// TIA Portal V16 export
// export: Created 2023-03-29T11:03:22.8937911Z, ExportSetting WithDefaults, DisplayName Totally Integrated Automation Portal, DisplayVersion V16 Update 6, DisplayName TIA Portal Version Control Interface, DisplayVersion V16 Update 2, DisplayName TIA Portal Openness, DisplayVersion V16 Update 6, DisplayName STEP 7 Professional, DisplayVersion V16 Update 6, DisplayName STEP 7 Safety, DisplayVersion V16, DisplayName WinCC Advanced, DisplayVersion V16 Update 6
FUNCTION "Wybór_aktywnego_zbiornika" : Void   // FC20, LAD
TITLE = Compressor selection from hours
{ S7_Optimized_Access := 'TRUE' }
AUTHOR : rtecmer
VERSION : 0.1
// Ustawienie kolejności wyboru zbiornika z wyrównaniem czasu pracy. Podstawa najmniejsza ilość godzin pracy
// stored: AutoNumber true, IsIECCheckEnabled false, SetENOAutomatically false, UDAEnableTagReadback false
   VAR_INPUT
      aktywny_Zbiornik_1 : Bool;   // zbiornik aktywny zasuwy na pozycji atomat
      aktywny_Zbiornik_2 : Bool;
      aktywny_Zbiornik_3 : Bool;
      aktywny_Zbiornik_4 : Bool;
      ready_Z1 : Bool;   // gotowość
      ready_Z2 : Bool;   // gotowość
      ready_Z3 : Bool;   // gotowość
      ready_Z4 : Bool;   // gotowość
      ready_Z5 : Bool;   // gotowość
      ready_Z6 : Bool;   // gotowość
      ready_Z7 : Bool;   // gotowość
      ready_Z8 : Bool;   // gotowość
      Is_Eptying : Bool;   // aktwny cykl napełniania
      Is_Filling : Bool;   // aktywny cykl pompownia
   END_VAR
   VAR_IN_OUT
      Reset : Bool;   // Reset po błędzie
      set_HWork_Tank_1 : Bool;   // ustawiony aktywny
      set_HWork_Tank_2 : Bool;   // ustawiony aktywny
      set_HWork_Tank_3 : Bool;   // ustawiony aktywny
      set_HWork_Tank_4 : Bool;   // ustawiony aktywny
      blok_tank_1 : Bool;   // blokowanie zbirnika w sekwencji
      blok_tank_2 : Bool;   // blokowanie zbirnika w sekwencji
      blok_tank_3 : Bool;   // blokowanie zbirnika w sekwencji
      blok_tank_4 : Bool;   // blokowanie zbirnika w sekwencji
   END_VAR
   VAR_TEMP
      tmp_Sum_sek_P1 : Real;
      tmp_Sum_sek_P2 : Real;
      tmp_Sum_sek_P3 : Real;
      tmp_Sum_sek_P4 : Real;
   END_VAR
BEGIN

REGION Network 1: Reakcja na równe liczniki
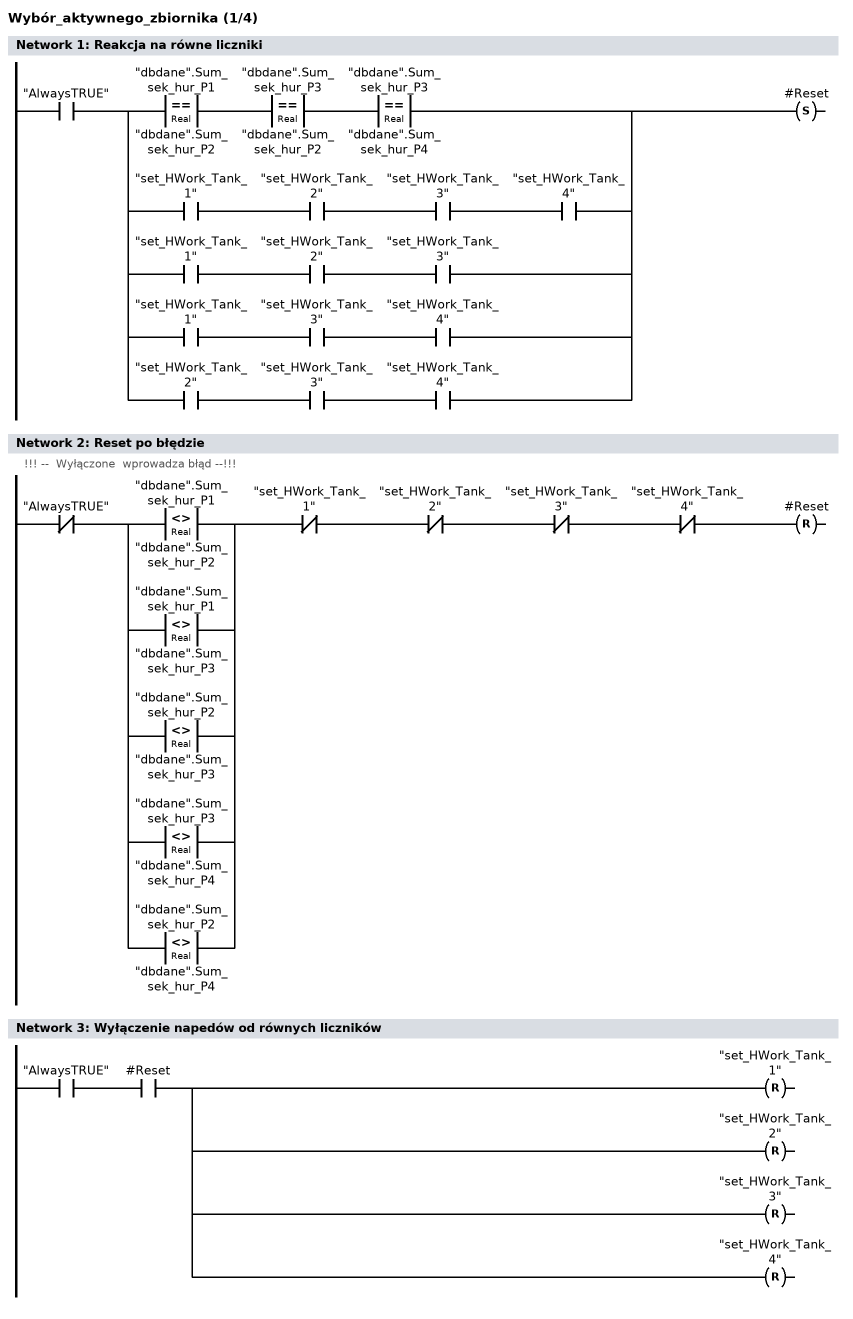
   RUNG wire#powerrail
      Contact( "AlwaysTRUE" )
      wire#w1
      { S7_Templates := "SrcType := Real" } EQ_Contact(in1 := "dbdane".Sum_sek_hur_P1, in2 := "dbdane".Sum_sek_hur_P2)
      { S7_Templates := "SrcType := Real" } EQ_Contact(in1 := "dbdane".Sum_sek_hur_P3, in2 := "dbdane".Sum_sek_hur_P2)
      { S7_Templates := "SrcType := Real" } EQ_Contact(in1 := "dbdane".Sum_sek_hur_P3, in2 := "dbdane".Sum_sek_hur_P4)
      wire#w2
      S_Coil( #Reset )
   END_RUNG
   RUNG wire#w1
      Contact( "set_HWork_Tank_1" )
      Contact( "set_HWork_Tank_2" )
      Contact( "set_HWork_Tank_3" )
      Contact( "set_HWork_Tank_4" )
   END_RUNG wire#w2
   RUNG wire#w1
      Contact( "set_HWork_Tank_1" )
      Contact( "set_HWork_Tank_2" )
      Contact( "set_HWork_Tank_3" )
   END_RUNG wire#w2
   RUNG wire#w1
      Contact( "set_HWork_Tank_1" )
      Contact( "set_HWork_Tank_3" )
      Contact( "set_HWork_Tank_4" )
   END_RUNG wire#w2
   RUNG wire#w1
      Contact( "set_HWork_Tank_2" )
      Contact( "set_HWork_Tank_3" )
      Contact( "set_HWork_Tank_4" )
   END_RUNG wire#w2
   // the same network as SCL:
   IF "AlwaysTRUE" AND ((("dbdane".Sum_sek_hur_P1 = "dbdane".Sum_sek_hur_P2) AND ("dbdane".Sum_sek_hur_P3 = "dbdane".Sum_sek_hur_P2) AND ("dbdane".Sum_sek_hur_P3 = "dbdane".Sum_sek_hur_P4)) OR ("set_HWork_Tank_1" AND "set_HWork_Tank_2" AND "set_HWork_Tank_3" AND "set_HWork_Tank_4") OR ("set_HWork_Tank_1" AND "set_HWork_Tank_2" AND "set_HWork_Tank_3") OR ("set_HWork_Tank_1" AND "set_HWork_Tank_3" AND "set_HWork_Tank_4") OR ("set_HWork_Tank_2" AND "set_HWork_Tank_3" AND "set_HWork_Tank_4")) THEN
       #Reset := TRUE;
   END_IF;
END_REGION

REGION Network 2: Reset po błędzie
   // !!! --  Wyłączone  wprowadza błąd --!!!
   RUNG wire#powerrail
      I_Contact( "AlwaysTRUE" )
      wire#w1
      { S7_Templates := "SrcType := Real" } NE_Contact(in1 := "dbdane".Sum_sek_hur_P1, in2 := "dbdane".Sum_sek_hur_P2)
      wire#w2
      I_Contact( "set_HWork_Tank_1" )
      I_Contact( "set_HWork_Tank_2" )
      I_Contact( "set_HWork_Tank_3" )
      I_Contact( "set_HWork_Tank_4" )
      R_Coil( #Reset )
   END_RUNG
   RUNG wire#w1
      { S7_Templates := "SrcType := Real" } NE_Contact(in1 := "dbdane".Sum_sek_hur_P1, in2 := "dbdane".Sum_sek_hur_P3)
   END_RUNG wire#w2
   RUNG wire#w1
      { S7_Templates := "SrcType := Real" } NE_Contact(in1 := "dbdane".Sum_sek_hur_P2, in2 := "dbdane".Sum_sek_hur_P3)
   END_RUNG wire#w2
   RUNG wire#w1
      { S7_Templates := "SrcType := Real" } NE_Contact(in1 := "dbdane".Sum_sek_hur_P3, in2 := "dbdane".Sum_sek_hur_P4)
   END_RUNG wire#w2
   RUNG wire#w1
      { S7_Templates := "SrcType := Real" } NE_Contact(in1 := "dbdane".Sum_sek_hur_P2, in2 := "dbdane".Sum_sek_hur_P4)
   END_RUNG wire#w2
   // the same network as SCL:
   IF NOT "AlwaysTRUE" AND (("dbdane".Sum_sek_hur_P1 <> "dbdane".Sum_sek_hur_P2) OR ("dbdane".Sum_sek_hur_P1 <> "dbdane".Sum_sek_hur_P3) OR ("dbdane".Sum_sek_hur_P2 <> "dbdane".Sum_sek_hur_P3) OR ("dbdane".Sum_sek_hur_P3 <> "dbdane".Sum_sek_hur_P4) OR ("dbdane".Sum_sek_hur_P2 <> "dbdane".Sum_sek_hur_P4)) AND NOT "set_HWork_Tank_1" AND NOT "set_HWork_Tank_2" AND NOT "set_HWork_Tank_3" AND NOT "set_HWork_Tank_4" THEN
       #Reset := FALSE;
   END_IF;
END_REGION

REGION Network 3: Wyłączenie napedów od równych liczników
   RUNG wire#powerrail
      Contact( "AlwaysTRUE" )
      Contact( #Reset )
      wire#w1
      R_Coil( "set_HWork_Tank_1" )
   END_RUNG
   RUNG wire#w1
      R_Coil( "set_HWork_Tank_2" )
   END_RUNG
   RUNG wire#w1
      R_Coil( "set_HWork_Tank_3" )
   END_RUNG
   RUNG wire#w1
      R_Coil( "set_HWork_Tank_4" )
   END_RUNG
   // the same network as SCL:
   IF "AlwaysTRUE" AND #Reset THEN
       "set_HWork_Tank_1" := FALSE;
       "set_HWork_Tank_2" := FALSE;
       "set_HWork_Tank_3" := FALSE;
       "set_HWork_Tank_4" := FALSE;
   END_IF;
END_REGION

REGION Network 4: Ustawienie domyślnych liczników startowych
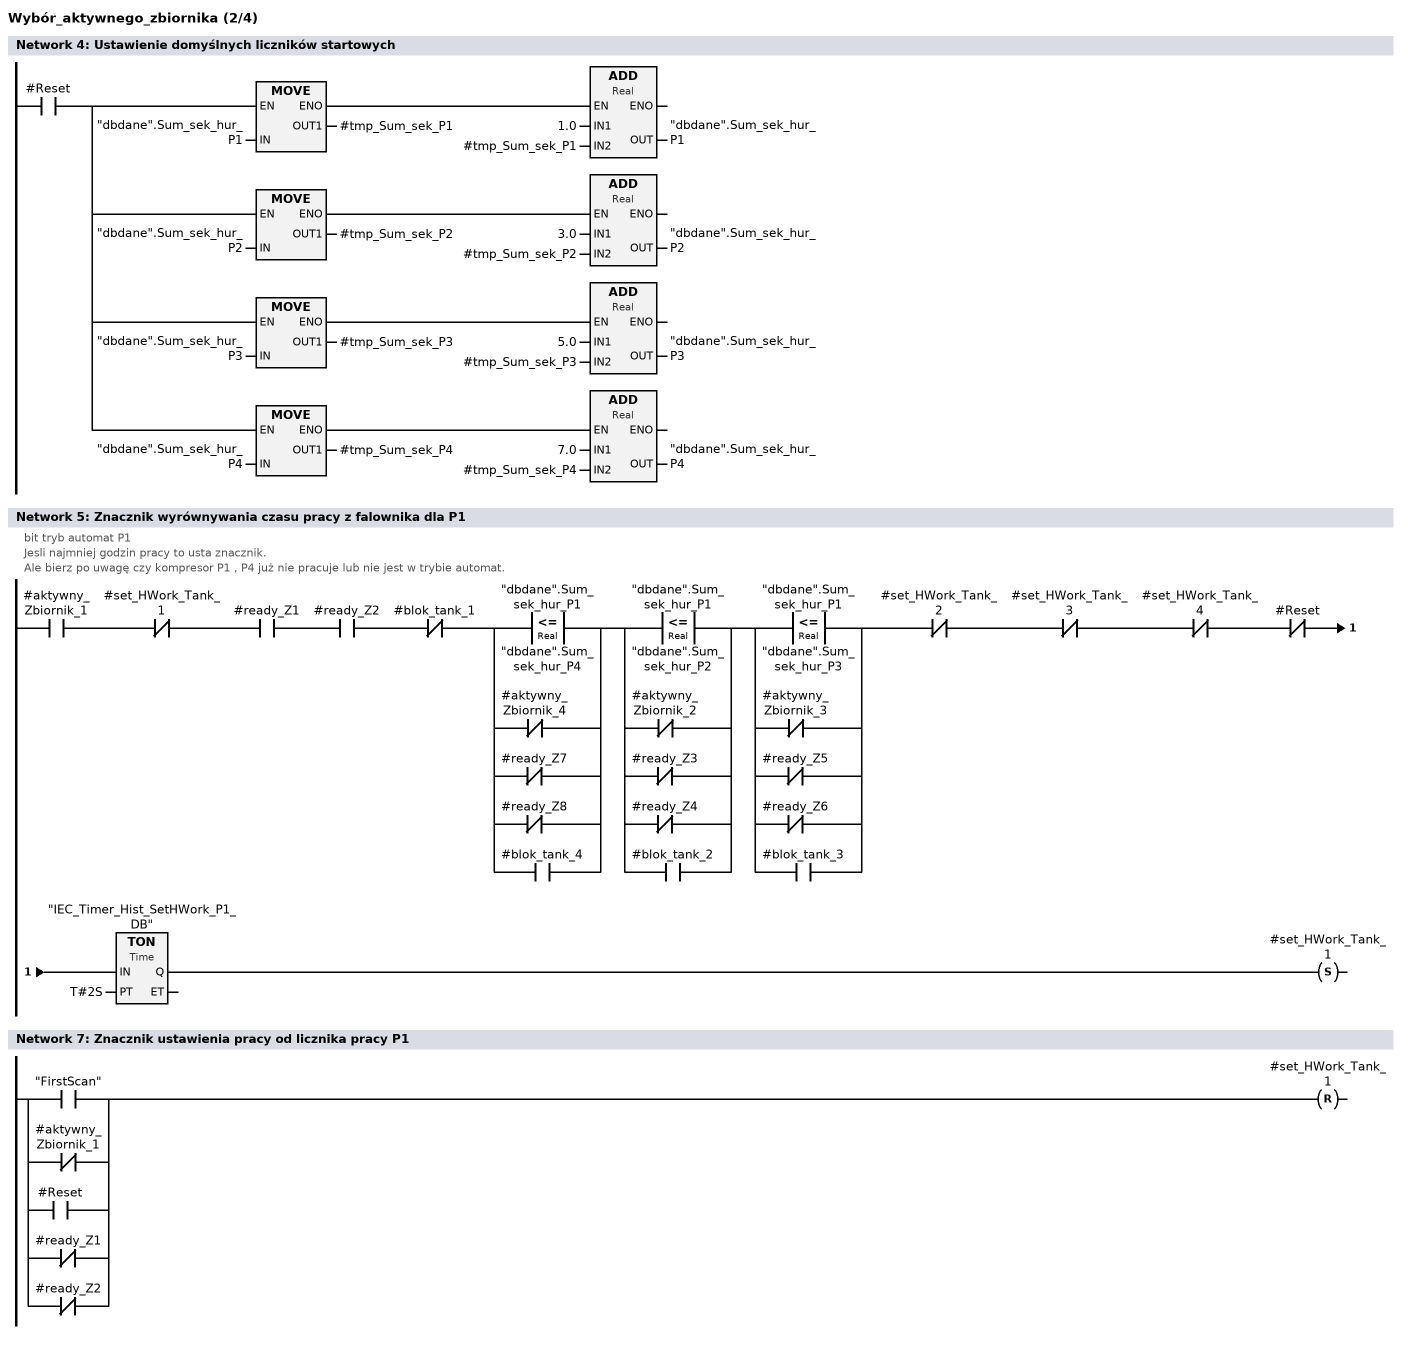
   RUNG wire#powerrail
      Contact( #Reset )
      wire#w1
      Move(in := "dbdane".Sum_sek_hur_P1, out1 => #tmp_Sum_sek_P1)
      { S7_Templates := "SrcType := Real" } Add(in1 := 1.0, in2 := #tmp_Sum_sek_P1, out => "dbdane".Sum_sek_hur_P1)
   END_RUNG
   RUNG wire#w1
      Move(in := "dbdane".Sum_sek_hur_P2, out1 => #tmp_Sum_sek_P2)
      { S7_Templates := "SrcType := Real" } Add(in1 := 3.0, in2 := #tmp_Sum_sek_P2, out => "dbdane".Sum_sek_hur_P2)
   END_RUNG
   RUNG wire#w1
      Move(in := "dbdane".Sum_sek_hur_P3, out1 => #tmp_Sum_sek_P3)
      { S7_Templates := "SrcType := Real" } Add(in1 := 5.0, in2 := #tmp_Sum_sek_P3, out => "dbdane".Sum_sek_hur_P3)
   END_RUNG
   RUNG wire#w1
      Move(in := "dbdane".Sum_sek_hur_P4, out1 => #tmp_Sum_sek_P4)
      { S7_Templates := "SrcType := Real" } Add(in1 := 7.0, in2 := #tmp_Sum_sek_P4, out => "dbdane".Sum_sek_hur_P4)
   END_RUNG
   // the same network as SCL:
   IF #Reset THEN
       #tmp_Sum_sek_P1 := "dbdane".Sum_sek_hur_P1;
       "dbdane".Sum_sek_hur_P1 := 1.0 + #tmp_Sum_sek_P1;
       #tmp_Sum_sek_P2 := "dbdane".Sum_sek_hur_P2;
       "dbdane".Sum_sek_hur_P2 := 3.0 + #tmp_Sum_sek_P2;
       #tmp_Sum_sek_P3 := "dbdane".Sum_sek_hur_P3;
       "dbdane".Sum_sek_hur_P3 := 5.0 + #tmp_Sum_sek_P3;
       #tmp_Sum_sek_P4 := "dbdane".Sum_sek_hur_P4;
       "dbdane".Sum_sek_hur_P4 := 7.0 + #tmp_Sum_sek_P4;
   END_IF;
END_REGION

REGION Network 5: Znacznik wyrównywania czasu pracy z falownika dla P1
   // bit tryb automat P1
   // Jesli najmniej godzin pracy to usta znacznik.
   // Ale bierz po uwagę czy kompresor P1 , P4 już nie pracuje lub nie jest w trybie automat.
   RUNG wire#powerrail
      Contact( #aktywny_Zbiornik_1 )
      I_Contact( #set_HWork_Tank_1 )
      Contact( #ready_Z1 )
      Contact( #ready_Z2 )
      I_Contact( #blok_tank_1 )
      wire#w1
      { S7_Templates := "SrcType := Real" } LE_Contact(in1 := "dbdane".Sum_sek_hur_P1, in2 := "dbdane".Sum_sek_hur_P4)
      wire#w2
      { S7_Templates := "SrcType := Real" } LE_Contact(in1 := "dbdane".Sum_sek_hur_P1, in2 := "dbdane".Sum_sek_hur_P2)
      wire#w3
      { S7_Templates := "SrcType := Real" } LE_Contact(in1 := "dbdane".Sum_sek_hur_P1, in2 := "dbdane".Sum_sek_hur_P3)
      wire#w4
      I_Contact( #set_HWork_Tank_2 )
      I_Contact( #set_HWork_Tank_3 )
      I_Contact( #set_HWork_Tank_4 )
      I_Contact( #Reset )
      { S7_Templates := "time_type := Time" } "IEC_Timer_Hist_SetHWork_P1_DB".TON(pt := T#2S, et =>)
      S_Coil( #set_HWork_Tank_1 )
   END_RUNG
   RUNG wire#w1
      I_Contact( #aktywny_Zbiornik_4 )
   END_RUNG wire#w2
   RUNG wire#w1
      I_Contact( #ready_Z7 )
   END_RUNG wire#w2
   RUNG wire#w1
      I_Contact( #ready_Z8 )
   END_RUNG wire#w2
   RUNG wire#w1
      Contact( #blok_tank_4 )
   END_RUNG wire#w2
   RUNG wire#w2
      I_Contact( #aktywny_Zbiornik_2 )
   END_RUNG wire#w3
   RUNG wire#w2
      I_Contact( #ready_Z3 )
   END_RUNG wire#w3
   RUNG wire#w2
      I_Contact( #ready_Z4 )
   END_RUNG wire#w3
   RUNG wire#w2
      Contact( #blok_tank_2 )
   END_RUNG wire#w3
   RUNG wire#w3
      I_Contact( #aktywny_Zbiornik_3 )
   END_RUNG wire#w4
   RUNG wire#w3
      I_Contact( #ready_Z5 )
   END_RUNG wire#w4
   RUNG wire#w3
      I_Contact( #ready_Z6 )
   END_RUNG wire#w4
   RUNG wire#w3
      Contact( #blok_tank_3 )
   END_RUNG wire#w4
   // the same network as SCL:
   "IEC_Timer_Hist_SetHWork_P1_DB".TON(IN := #aktywny_Zbiornik_1 AND NOT #set_HWork_Tank_1 AND #ready_Z1 AND #ready_Z2 AND NOT #blok_tank_1 AND (("dbdane".Sum_sek_hur_P1 <= "dbdane".Sum_sek_hur_P4) OR NOT #aktywny_Zbiornik_4 OR NOT #ready_Z7 OR NOT #ready_Z8 OR #blok_tank_4) AND (("dbdane".Sum_sek_hur_P1 <= "dbdane".Sum_sek_hur_P2) OR NOT #aktywny_Zbiornik_2 OR NOT #ready_Z3 OR NOT #ready_Z4 OR #blok_tank_2) AND (("dbdane".Sum_sek_hur_P1 <= "dbdane".Sum_sek_hur_P3) OR NOT #aktywny_Zbiornik_3 OR NOT #ready_Z5 OR NOT #ready_Z6 OR #blok_tank_3) AND NOT #set_HWork_Tank_2 AND NOT #set_HWork_Tank_3 AND NOT #set_HWork_Tank_4 AND NOT #Reset,
                           PT := T#2S);
   IF "IEC_Timer_Hist_SetHWork_P1_DB".Q THEN #set_HWork_Tank_1 := TRUE; END_IF;
END_REGION

REGION Network 6 (SCL): Sprawdzanie czy aktywna w trybie AUT
   IF "set_HWork_Tank_1" = TRUE AND #aktywny_Zbiornik_1 = FALSE THEN
     // Statement section IF
     "set_HWork_Tank_1" := FALSE;
     ;
   END_IF;
END_REGION

REGION Network 7: Znacznik ustawienia pracy od licznika pracy P1
   RUNG wire#powerrail
      Contact( "FirstScan" )
      wire#w1
      R_Coil( #set_HWork_Tank_1 )
   END_RUNG
   RUNG wire#powerrail
      I_Contact( #aktywny_Zbiornik_1 )
   END_RUNG wire#w1
   RUNG wire#powerrail
      Contact( #Reset )
   END_RUNG wire#w1
   RUNG wire#powerrail
      I_Contact( #ready_Z1 )
   END_RUNG wire#w1
   RUNG wire#powerrail
      I_Contact( #ready_Z2 )
   END_RUNG wire#w1
   // the same network as SCL:
   IF "FirstScan" OR NOT #aktywny_Zbiornik_1 OR #Reset OR NOT #ready_Z1 OR NOT #ready_Z2 THEN
       #set_HWork_Tank_1 := FALSE;
   END_IF;
END_REGION

REGION Network 8: Znacznik wyrównywania czasu pracy z falownika dla P2
   // %DB10.DBX9.7 - bit tryb automat P2
   // Jesli najmniej godzin pracy to usta znacznik.
   // Ale bierz po uwagę czy kompresor P1 , P4 już nie pracuje lub nie jest w trybie automat.
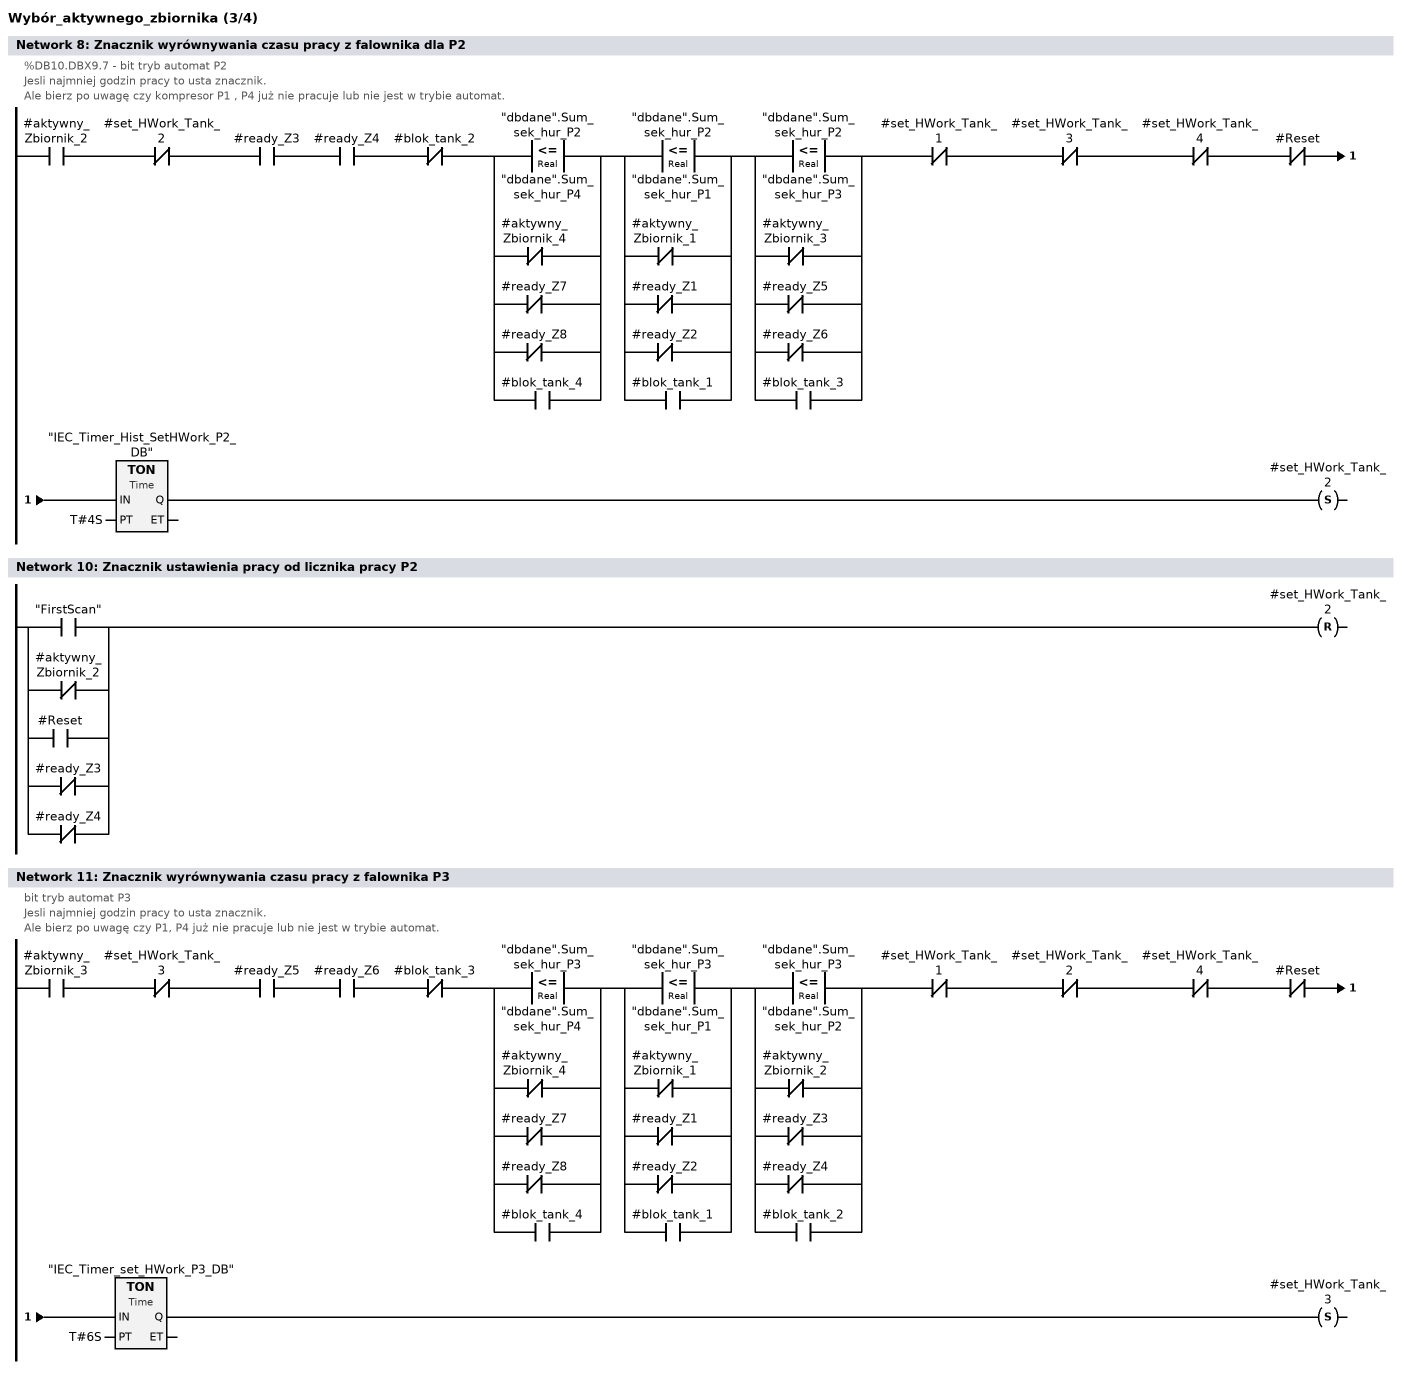
   RUNG wire#powerrail
      Contact( #aktywny_Zbiornik_2 )
      I_Contact( #set_HWork_Tank_2 )
      Contact( #ready_Z3 )
      Contact( #ready_Z4 )
      I_Contact( #blok_tank_2 )
      wire#w1
      { S7_Templates := "SrcType := Real" } LE_Contact(in1 := "dbdane".Sum_sek_hur_P2, in2 := "dbdane".Sum_sek_hur_P4)
      wire#w2
      { S7_Templates := "SrcType := Real" } LE_Contact(in1 := "dbdane".Sum_sek_hur_P2, in2 := "dbdane".Sum_sek_hur_P1)
      wire#w3
      { S7_Templates := "SrcType := Real" } LE_Contact(in1 := "dbdane".Sum_sek_hur_P2, in2 := "dbdane".Sum_sek_hur_P3)
      wire#w4
      I_Contact( #set_HWork_Tank_1 )
      I_Contact( #set_HWork_Tank_3 )
      I_Contact( #set_HWork_Tank_4 )
      I_Contact( #Reset )
      { S7_Templates := "time_type := Time" } "IEC_Timer_Hist_SetHWork_P2_DB".TON(pt := T#4S, et =>)
      S_Coil( #set_HWork_Tank_2 )
   END_RUNG
   RUNG wire#w1
      I_Contact( #aktywny_Zbiornik_4 )
   END_RUNG wire#w2
   RUNG wire#w1
      I_Contact( #ready_Z7 )
   END_RUNG wire#w2
   RUNG wire#w1
      I_Contact( #ready_Z8 )
   END_RUNG wire#w2
   RUNG wire#w1
      Contact( #blok_tank_4 )
   END_RUNG wire#w2
   RUNG wire#w2
      I_Contact( #aktywny_Zbiornik_1 )
   END_RUNG wire#w3
   RUNG wire#w2
      I_Contact( #ready_Z1 )
   END_RUNG wire#w3
   RUNG wire#w2
      I_Contact( #ready_Z2 )
   END_RUNG wire#w3
   RUNG wire#w2
      Contact( #blok_tank_1 )
   END_RUNG wire#w3
   RUNG wire#w3
      I_Contact( #aktywny_Zbiornik_3 )
   END_RUNG wire#w4
   RUNG wire#w3
      I_Contact( #ready_Z5 )
   END_RUNG wire#w4
   RUNG wire#w3
      I_Contact( #ready_Z6 )
   END_RUNG wire#w4
   RUNG wire#w3
      Contact( #blok_tank_3 )
   END_RUNG wire#w4
   // the same network as SCL:
   "IEC_Timer_Hist_SetHWork_P2_DB".TON(IN := #aktywny_Zbiornik_2 AND NOT #set_HWork_Tank_2 AND #ready_Z3 AND #ready_Z4 AND NOT #blok_tank_2 AND (("dbdane".Sum_sek_hur_P2 <= "dbdane".Sum_sek_hur_P4) OR NOT #aktywny_Zbiornik_4 OR NOT #ready_Z7 OR NOT #ready_Z8 OR #blok_tank_4) AND (("dbdane".Sum_sek_hur_P2 <= "dbdane".Sum_sek_hur_P1) OR NOT #aktywny_Zbiornik_1 OR NOT #ready_Z1 OR NOT #ready_Z2 OR #blok_tank_1) AND (("dbdane".Sum_sek_hur_P2 <= "dbdane".Sum_sek_hur_P3) OR NOT #aktywny_Zbiornik_3 OR NOT #ready_Z5 OR NOT #ready_Z6 OR #blok_tank_3) AND NOT #set_HWork_Tank_1 AND NOT #set_HWork_Tank_3 AND NOT #set_HWork_Tank_4 AND NOT #Reset,
                           PT := T#4S);
   IF "IEC_Timer_Hist_SetHWork_P2_DB".Q THEN #set_HWork_Tank_2 := TRUE; END_IF;
END_REGION

REGION Network 9 (SCL): Sprawdzanie czy aktywna w trybie AUT
   IF "set_HWork_Tank_2" = TRUE AND #aktywny_Zbiornik_2 = FALSE THEN
     // Statement section IF
     "set_HWork_Tank_2" := FALSE;
     ;
   END_IF;
END_REGION

REGION Network 10: Znacznik ustawienia pracy od licznika pracy P2
   RUNG wire#powerrail
      Contact( "FirstScan" )
      wire#w1
      R_Coil( #set_HWork_Tank_2 )
   END_RUNG
   RUNG wire#powerrail
      I_Contact( #aktywny_Zbiornik_2 )
   END_RUNG wire#w1
   RUNG wire#powerrail
      Contact( #Reset )
   END_RUNG wire#w1
   RUNG wire#powerrail
      I_Contact( #ready_Z3 )
   END_RUNG wire#w1
   RUNG wire#powerrail
      I_Contact( #ready_Z4 )
   END_RUNG wire#w1
   // the same network as SCL:
   IF "FirstScan" OR NOT #aktywny_Zbiornik_2 OR #Reset OR NOT #ready_Z3 OR NOT #ready_Z4 THEN
       #set_HWork_Tank_2 := FALSE;
   END_IF;
END_REGION

REGION Network 11: Znacznik wyrównywania czasu pracy z falownika P3
   // bit tryb automat P3
   // Jesli najmniej godzin pracy to usta znacznik.
   // Ale bierz po uwagę czy P1, P4 już nie pracuje lub nie jest w trybie automat.
   RUNG wire#powerrail
      Contact( #aktywny_Zbiornik_3 )
      I_Contact( #set_HWork_Tank_3 )
      Contact( #ready_Z5 )
      Contact( #ready_Z6 )
      I_Contact( #blok_tank_3 )
      wire#w1
      { S7_Templates := "SrcType := Real" } LE_Contact(in1 := "dbdane".Sum_sek_hur_P3, in2 := "dbdane".Sum_sek_hur_P4)
      wire#w2
      { S7_Templates := "SrcType := Real" } LE_Contact(in1 := "dbdane".Sum_sek_hur_P3, in2 := "dbdane".Sum_sek_hur_P1)
      wire#w3
      { S7_Templates := "SrcType := Real" } LE_Contact(in1 := "dbdane".Sum_sek_hur_P3, in2 := "dbdane".Sum_sek_hur_P2)
      wire#w4
      I_Contact( #set_HWork_Tank_1 )
      I_Contact( #set_HWork_Tank_2 )
      I_Contact( #set_HWork_Tank_4 )
      I_Contact( #Reset )
      { S7_Templates := "time_type := Time" } "IEC_Timer_set_HWork_P3_DB".TON(pt := T#6S, et =>)
      S_Coil( #set_HWork_Tank_3 )
   END_RUNG
   RUNG wire#w1
      I_Contact( #aktywny_Zbiornik_4 )
   END_RUNG wire#w2
   RUNG wire#w1
      I_Contact( #ready_Z7 )
   END_RUNG wire#w2
   RUNG wire#w1
      I_Contact( #ready_Z8 )
   END_RUNG wire#w2
   RUNG wire#w1
      Contact( #blok_tank_4 )
   END_RUNG wire#w2
   RUNG wire#w2
      I_Contact( #aktywny_Zbiornik_1 )
   END_RUNG wire#w3
   RUNG wire#w2
      I_Contact( #ready_Z1 )
   END_RUNG wire#w3
   RUNG wire#w2
      I_Contact( #ready_Z2 )
   END_RUNG wire#w3
   RUNG wire#w2
      Contact( #blok_tank_1 )
   END_RUNG wire#w3
   RUNG wire#w3
      I_Contact( #aktywny_Zbiornik_2 )
   END_RUNG wire#w4
   RUNG wire#w3
      I_Contact( #ready_Z3 )
   END_RUNG wire#w4
   RUNG wire#w3
      I_Contact( #ready_Z4 )
   END_RUNG wire#w4
   RUNG wire#w3
      Contact( #blok_tank_2 )
   END_RUNG wire#w4
   // the same network as SCL:
   "IEC_Timer_set_HWork_P3_DB".TON(IN := #aktywny_Zbiornik_3 AND NOT #set_HWork_Tank_3 AND #ready_Z5 AND #ready_Z6 AND NOT #blok_tank_3 AND (("dbdane".Sum_sek_hur_P3 <= "dbdane".Sum_sek_hur_P4) OR NOT #aktywny_Zbiornik_4 OR NOT #ready_Z7 OR NOT #ready_Z8 OR #blok_tank_4) AND (("dbdane".Sum_sek_hur_P3 <= "dbdane".Sum_sek_hur_P1) OR NOT #aktywny_Zbiornik_1 OR NOT #ready_Z1 OR NOT #ready_Z2 OR #blok_tank_1) AND (("dbdane".Sum_sek_hur_P3 <= "dbdane".Sum_sek_hur_P2) OR NOT #aktywny_Zbiornik_2 OR NOT #ready_Z3 OR NOT #ready_Z4 OR #blok_tank_2) AND NOT #set_HWork_Tank_1 AND NOT #set_HWork_Tank_2 AND NOT #set_HWork_Tank_4 AND NOT #Reset,
                           PT := T#6S);
   IF "IEC_Timer_set_HWork_P3_DB".Q THEN #set_HWork_Tank_3 := TRUE; END_IF;
END_REGION

REGION Network 12 (SCL): Sprawdzanie czy aktywna w trybie AUT
   IF "set_HWork_Tank_3" = TRUE AND #aktywny_Zbiornik_3 = FALSE THEN
     // Statement section IF
     "set_HWork_Tank_3":= FALSE;
     ;
   END_IF;
END_REGION

REGION Network 13: Znacznik ustawienia pracy od licznika pracy P3
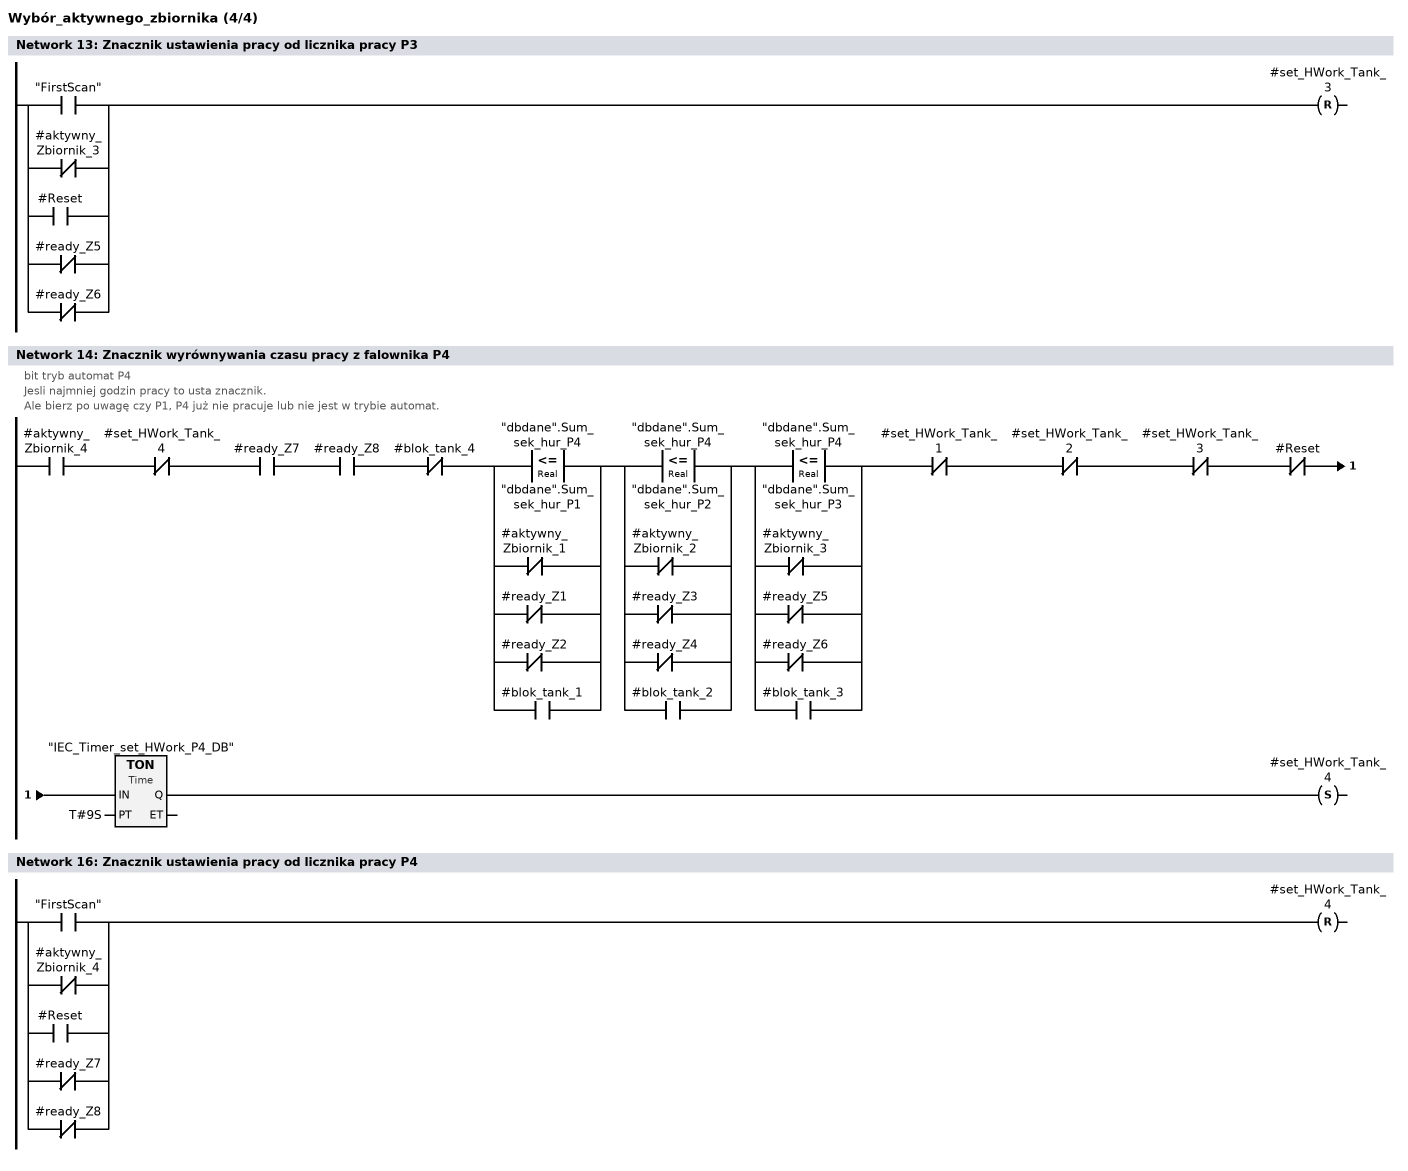
   RUNG wire#powerrail
      Contact( "FirstScan" )
      wire#w1
      R_Coil( #set_HWork_Tank_3 )
   END_RUNG
   RUNG wire#powerrail
      I_Contact( #aktywny_Zbiornik_3 )
   END_RUNG wire#w1
   RUNG wire#powerrail
      Contact( #Reset )
   END_RUNG wire#w1
   RUNG wire#powerrail
      I_Contact( #ready_Z5 )
   END_RUNG wire#w1
   RUNG wire#powerrail
      I_Contact( #ready_Z6 )
   END_RUNG wire#w1
   // the same network as SCL:
   IF "FirstScan" OR NOT #aktywny_Zbiornik_3 OR #Reset OR NOT #ready_Z5 OR NOT #ready_Z6 THEN
       #set_HWork_Tank_3 := FALSE;
   END_IF;
END_REGION

REGION Network 14: Znacznik wyrównywania czasu pracy z falownika P4
   // bit tryb automat P4
   // Jesli najmniej godzin pracy to usta znacznik.
   // Ale bierz po uwagę czy P1, P4 już nie pracuje lub nie jest w trybie automat.
   RUNG wire#powerrail
      Contact( #aktywny_Zbiornik_4 )
      I_Contact( #set_HWork_Tank_4 )
      Contact( #ready_Z7 )
      Contact( #ready_Z8 )
      I_Contact( #blok_tank_4 )
      wire#w1
      { S7_Templates := "SrcType := Real" } LE_Contact(in1 := "dbdane".Sum_sek_hur_P4, in2 := "dbdane".Sum_sek_hur_P1)
      wire#w2
      { S7_Templates := "SrcType := Real" } LE_Contact(in1 := "dbdane".Sum_sek_hur_P4, in2 := "dbdane".Sum_sek_hur_P2)
      wire#w3
      { S7_Templates := "SrcType := Real" } LE_Contact(in1 := "dbdane".Sum_sek_hur_P4, in2 := "dbdane".Sum_sek_hur_P3)
      wire#w4
      I_Contact( #set_HWork_Tank_1 )
      I_Contact( #set_HWork_Tank_2 )
      I_Contact( #set_HWork_Tank_3 )
      I_Contact( #Reset )
      { S7_Templates := "time_type := Time" } "IEC_Timer_set_HWork_P4_DB".TON(pt := T#9S, et =>)
      S_Coil( #set_HWork_Tank_4 )
   END_RUNG
   RUNG wire#w1
      I_Contact( #aktywny_Zbiornik_1 )
   END_RUNG wire#w2
   RUNG wire#w1
      I_Contact( #ready_Z1 )
   END_RUNG wire#w2
   RUNG wire#w1
      I_Contact( #ready_Z2 )
   END_RUNG wire#w2
   RUNG wire#w1
      Contact( #blok_tank_1 )
   END_RUNG wire#w2
   RUNG wire#w2
      I_Contact( #aktywny_Zbiornik_2 )
   END_RUNG wire#w3
   RUNG wire#w2
      I_Contact( #ready_Z3 )
   END_RUNG wire#w3
   RUNG wire#w2
      I_Contact( #ready_Z4 )
   END_RUNG wire#w3
   RUNG wire#w2
      Contact( #blok_tank_2 )
   END_RUNG wire#w3
   RUNG wire#w3
      I_Contact( #aktywny_Zbiornik_3 )
   END_RUNG wire#w4
   RUNG wire#w3
      I_Contact( #ready_Z5 )
   END_RUNG wire#w4
   RUNG wire#w3
      I_Contact( #ready_Z6 )
   END_RUNG wire#w4
   RUNG wire#w3
      Contact( #blok_tank_3 )
   END_RUNG wire#w4
   // the same network as SCL:
   "IEC_Timer_set_HWork_P4_DB".TON(IN := #aktywny_Zbiornik_4 AND NOT #set_HWork_Tank_4 AND #ready_Z7 AND #ready_Z8 AND NOT #blok_tank_4 AND (("dbdane".Sum_sek_hur_P4 <= "dbdane".Sum_sek_hur_P1) OR NOT #aktywny_Zbiornik_1 OR NOT #ready_Z1 OR NOT #ready_Z2 OR #blok_tank_1) AND (("dbdane".Sum_sek_hur_P4 <= "dbdane".Sum_sek_hur_P2) OR NOT #aktywny_Zbiornik_2 OR NOT #ready_Z3 OR NOT #ready_Z4 OR #blok_tank_2) AND (("dbdane".Sum_sek_hur_P4 <= "dbdane".Sum_sek_hur_P3) OR NOT #aktywny_Zbiornik_3 OR NOT #ready_Z5 OR NOT #ready_Z6 OR #blok_tank_3) AND NOT #set_HWork_Tank_1 AND NOT #set_HWork_Tank_2 AND NOT #set_HWork_Tank_3 AND NOT #Reset,
                           PT := T#9S);
   IF "IEC_Timer_set_HWork_P4_DB".Q THEN #set_HWork_Tank_4 := TRUE; END_IF;
END_REGION

REGION Network 15 (SCL): Sprawdzanie czy aktywna w trybie AUT
   IF "set_HWork_Tank_4" = TRUE AND #aktywny_Zbiornik_4 = FALSE THEN
     // Statement section IF
     "set_HWork_Tank_4" := FALSE;
     ;
   END_IF;
END_REGION

REGION Network 16: Znacznik ustawienia pracy od licznika pracy P4
   RUNG wire#powerrail
      Contact( "FirstScan" )
      wire#w1
      R_Coil( #set_HWork_Tank_4 )
   END_RUNG
   RUNG wire#powerrail
      I_Contact( #aktywny_Zbiornik_4 )
   END_RUNG wire#w1
   RUNG wire#powerrail
      Contact( #Reset )
   END_RUNG wire#w1
   RUNG wire#powerrail
      I_Contact( #ready_Z7 )
   END_RUNG wire#w1
   RUNG wire#powerrail
      I_Contact( #ready_Z8 )
   END_RUNG wire#w1
   // the same network as SCL:
   IF "FirstScan" OR NOT #aktywny_Zbiornik_4 OR #Reset OR NOT #ready_Z7 OR NOT #ready_Z8 THEN
       #set_HWork_Tank_4 := FALSE;
   END_IF;
END_REGION
END_FUNCTION
